(* Schneider Machine Expert - Basic project Enkoder, file version 1.8.0.0 *)
(* ProjectInformations: Name=Yeni proje *)

HARDWARE
  Cpu 0: TM221ME16T/G
  ModuleExtensionObject 0: TM3DI8/G
  ModuleExtensionObject 1: TM3AQ2/G
  EthernetConfiguration: NetworkName=M221, IpAllocationMode=FixedAddress, IpAddress=192.168.0.15, SubnetMask=255.255.255.0
  SerialLineConfiguration: Baud=Baud19200, Parity=ParityNone, DataBits=DataBits8, StopBits=StopBits1, PhysicalMedium=PhysicalMediumRs485, TransmissionMode=TransmissionModeModbusRtu, SlaveId=1, Addressing=SlaveAddressing
  MastTask: UsePeriodScanMode=false, PeriodScan=100
  FastTask: Period=255
  CpuBehavior: StartingMode=StartAsPreviousState, AutoSaveRamOnEeprom=true, WatchdogPeriod=250

SYMBOLS  (address, symbol, comment, settings)
  %M0         "HMI/FIRÇA YUKARI"
  %M1         "HMI/FIRÇA AŞAĞI"
  %M2         "HMI/FIRÇA 2 YUKARI"
  %M3         "HMI/FIRÇA 2 AŞAĞI"
  %M4         "HMI BANT START"
  %M5         "HMI OSILASYON START"
  %M6         "427"
  %M7         "428"
  %I0.0       "403/FIRÇA1 ÜST SINIR ANAHTARI"
  %I0.1       "402/FIRÇA1 ALT SINIR ANAHTARI"
  %I0.2       "405/FIRÇA2/ÜST SINIR ANAHTARI"
  %I0.3       "404/FIRÇA2/ ALT SINIR ANAHTARI"
  %Q0.0       "421/FIRÇA YUKARI"
  %Q0.1       "422/FIRÇA AŞAĞI"
  %Q0.2       "423/FIRÇA 2 YUKARI"
  %Q0.3       "424/FIRÇA 2 AŞAĞI"
  %Q0.4       "425/BANT START"
  %Q0.5       "426/OSILASYON START"
  %Q0.6       "427"
  %Q0.7       "428"
  %HSC0       [Type=CounterOrDownCounterBiPhasesX4, Preset=0, ThresholdS0=1000, ThresholdS1=2000, DedicatedInputs(DedicatedInput(Activated=true), DedicatedInput(Activated=true)), ReflexOutputs(ReflexOutput(Activated=true, LessThanS0=false, GreaterOrEqualThanS0=true, GreaterOrEqualThanS1=false), ReflexOutput(Activated=true, LessThanS0=false, GreaterOrEqualThanS0=false, GreaterOrEqualThanS1=true)), Thresholds(Thre]

POU Yeni POU
  (* SectionNumber=1 *)

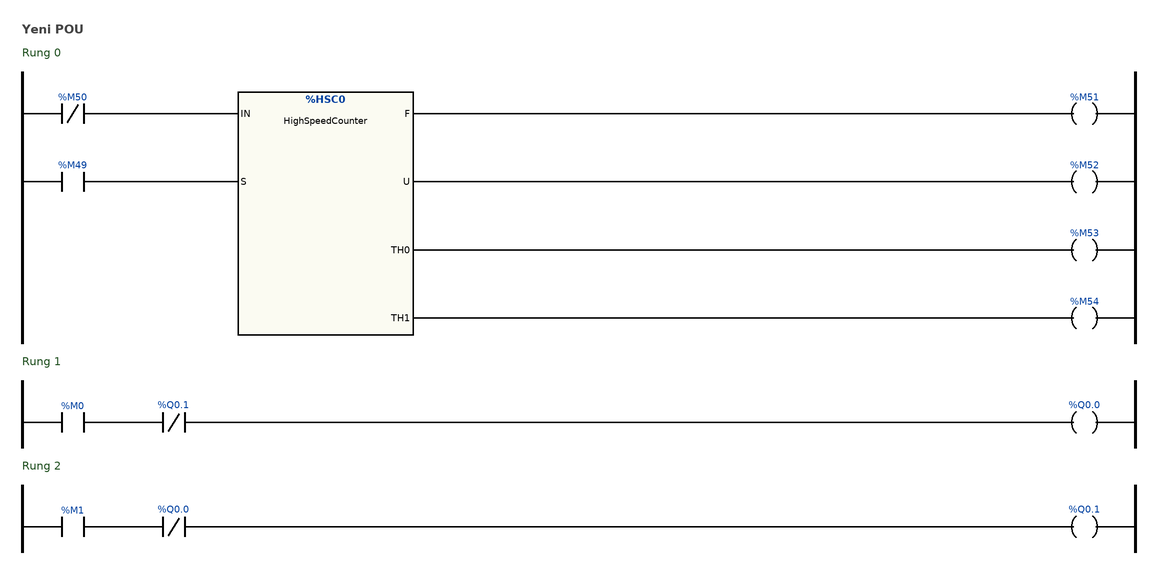

// Rung 0
  BLK %HSC0
  LDN %M50
  IN
  LD %M49
  S
  OUT_BLK
  LD F
  ST %M51
  LD U
  ST %M52
  LD TH0
  ST %M53
  LD TH1
  ST %M54
  END_BLK
  // as ST:
  //   %HSC0(IN := NOT %M50, S := %M49);
  //   %M51 := %HSC0.F;
  //   %M52 := %HSC0.U;
  //   %M53 := %HSC0.TH0;
  //   %M54 := %HSC0.TH1;

// Rung 1
  LD %M0
  ANDN %Q0.1
  ST %Q0.0
  // as ST:
  //   %Q0.0 := %M0 AND NOT %Q0.1;

// Rung 2
  LD %M1
  ANDN %Q0.0
  ST %Q0.1
  // as ST:
  //   %Q0.1 := %M1 AND NOT %Q0.0;
